SUBAPPLICATION Uebung_003c_sub (* IX auf QX (generisch) *)
  (* Standard: 61499-2; Description: Copyright (c) 2023 Meisterschulen am Ostbahnhof This program and the accompanying materials are made available under the terms of the Eclipse Public License 2.0 which is available at https://www.eclipse.org/legal/epl-2.0/ SPDX-License-Identifier: EPL-2.0 *)
  (* Version 1.0, 2023-10-23, Franz Höpfinger, Meisterschulen am Ostbahnhof *)
  PACKAGE Uebungen;
  IMPORT logiBUS::io::DI::logiBUS_DI::Invalid;
  IMPORT logiBUS::io::DI::logiBUS_DI_S;
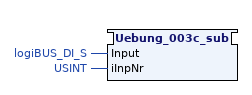
  VAR_INPUT
    Input : logiBUS::io::DI::logiBUS_DI_S := Invalid; (* Identify the Input Input_I1..I8 *)
    iInpNr : USINT := 0; (* Number of auxiliary array - corresponds with the order in the pool that means first aux input in pool is iInpNr = 0 etc. *)
  END_VAR
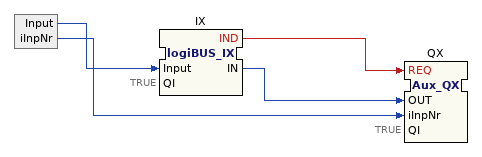
  FBS
    QX : Aux_QX(QI := TRUE);
    IX : logiBUS::io::DI::logiBUS_IX(QI := TRUE);
  END_FBS
  EVENT_CONNECTIONS
    IX.IND TO QX.REQ;
  END_CONNECTIONS
  DATA_CONNECTIONS
    IX.IN TO QX.OUT;
    Input TO IX.Input;
    iInpNr TO QX.iInpNr;
  END_CONNECTIONS
END_SUBAPPLICATION
